Fanuc KAREL source: kt00165.compact.KL

PROGRAM KT00165
%STACKSIZE=65535
%PRIORITY=65535
%NOLOCKGROUP
VAR
I1 : INTEGER
Y2 : ARRAY[2] OF BYTE
OUT : INTEGER
BEGIN
I1=2
Y2[1]=3
OUT=(I1 MOD Y2[1])
END KT00165
